// TIA Portal V20 export
// export: Created 2025-12-01T14:56:17.9021417Z, ExportSetting None, DisplayName Totally Integrated Automation Portal, DisplayVersion V20 Update 3, DisplayName TIA Portal Openness, DisplayVersion V20 Update 3, DisplayName TIA Portal Version Control Interface, DisplayVersion V20 Update 3, DisplayName STEP 7 Professional, DisplayVersion V20 Update 3, DisplayName STEP 7 Safety, DisplayVersion V20 Update 2, DisplayName WinCC Basic/Comfort/Advanced, DisplayVersion V20 Update 3, DisplayName WinCC Professional, DisplayVersion V20 Update 3, DisplayName WinCC Unified, DisplayVersion V20 Update 3
TYPE "Avisos_Mesa_HMI"
   STRUCT
      NoHayUT_EnMesa : Bool;
      RefrescoUT_EnMesa : Bool;
      UTMovidaConExito : Bool;
      Bit_03 : Bool;
      PeticionVisualizarMesa_OK : Bool;
      PeticionVisualizarMesa_SinMesaPedida : Bool;
      PeticionVisualizarMesa_Ocupada : Bool;
      PeticionVisualizarMesa_TOut : Bool;
      Bit_10 : Bool;
      Bit_11 : Bool;
      Bit_12 : Bool;
      Bit_13 : Bool;
      Bit_14 : Bool;
      Bit_15 : Bool;
      Clock_Comm : Bool;
      MemoKeepAlive : Bool;
   END_STRUCT;
END_TYPE
